INTERFACE I_KeyValueCollectionDisposedEvent EXTENDS I_Event

PROPERTY PUBLIC Target : I_KeyValueCollection
GET
END_GET
END_PROPERTY

END_INTERFACE

(* stored: Version 1.1.0.1, ProductVersion 3.1.4024.12
   Itf I_KeyValueCollectionDisposedEvent: Id {aa814d9a-6293-4505-9227-a52714cfd861}
   Property Target: Id {dccb2463-20f6-41a0-a100-dc30c563568b}
   Get Get: Id {73206542-689a-40c2-a172-263a06e61524} *)
